FUNCTION_BLOCK MulticastTwoConCtl (* Composite Function Block Type *)
  (* Standard: 61499-2 *)
  (* Version 0.2, 2003-12-05, JHC, Rockwell Automation, Renamed from NEWCOMPFB. *)
  (* Version 0.1, 2002-01-08, JHC, Rockwell Automation, Added DLY FB as example. *)
  (* Version 0.0, 2000-05-27, JHC, Rockwell Automation *)
  (* Compiler header: package fb.rt.cs725; *)
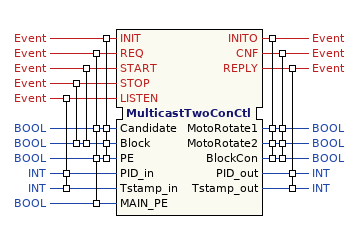
  EVENT_INPUT
    INIT WITH Candidate, Block, PE; (* Initialization Request *)
    REQ WITH Candidate, PE, MAIN_PE; (* Normal Execution Request *)
    START WITH Block;
    STOP WITH Block;
    LISTEN WITH Tstamp_in, PID_in;
  END_EVENT
  EVENT_OUTPUT
    INITO WITH MotoRotate1, MotoRotate2, BlockCon; (* Initialization Confirm *)
    CNF WITH MotoRotate1, MotoRotate2, BlockCon; (* Execution Confirmation *)
    REPLY WITH PID_out, Tstamp_out;
  END_EVENT
  VAR_INPUT
    Candidate : BOOL;
    Block : BOOL;
    PE : BOOL;
    PID_in : INT;
    Tstamp_in : INT;
    MAIN_PE : BOOL;
  END_VAR
  VAR_OUTPUT
    MotoRotate1 : BOOL;
    MotoRotate2 : BOOL;
    BlockCon : BOOL;
    PID_out : INT;
    Tstamp_out : INT;
  END_VAR
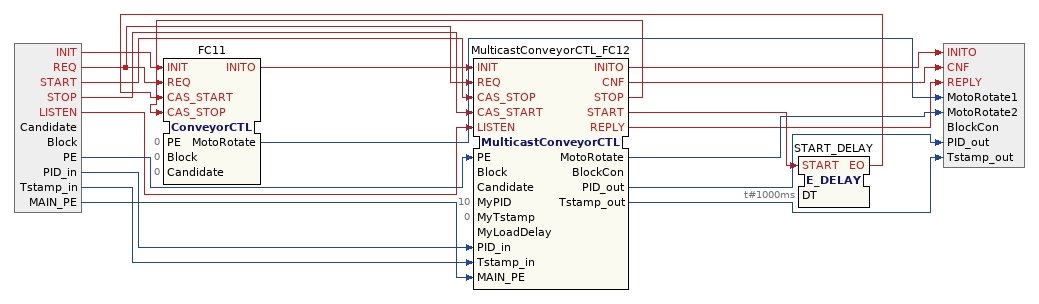
  FBS
    FC11 : ConveyorCTL(PE := 0, Block := 0, Candidate := 0);
    MulticastConveyorCTL_FC12 : MulticastConveyorCTL(MyPID := 10, MyTstamp := 0);
    START_DELAY : E_DELAY(DT := t#1000ms);
  END_FBS
  EVENT_CONNECTIONS
    INIT TO FC11.INIT;
    REQ TO FC11.REQ;
    LISTEN TO MulticastConveyorCTL_FC12.LISTEN;
    MulticastConveyorCTL_FC12.REPLY TO REPLY;
    FC11.INITO TO MulticastConveyorCTL_FC12.INIT;
    MulticastConveyorCTL_FC12.CNF TO CNF;
    MulticastConveyorCTL_FC12.INITO TO INITO;
    START TO MulticastConveyorCTL_FC12.CAS_STOP;
    STOP TO MulticastConveyorCTL_FC12.CAS_START;
    REQ TO MulticastConveyorCTL_FC12.REQ;
    MulticastConveyorCTL_FC12.START TO START_DELAY.START;
    START_DELAY.EO TO FC11.CAS_START;
    MulticastConveyorCTL_FC12.STOP TO FC11.CAS_STOP;
  END_CONNECTIONS
  DATA_CONNECTIONS
    FC11.MotoRotate TO MotoRotate1;
    PE TO MulticastConveyorCTL_FC12.PE;
    PID_in TO MulticastConveyorCTL_FC12.PID_in;
    Tstamp_in TO MulticastConveyorCTL_FC12.Tstamp_in;
    MulticastConveyorCTL_FC12.Tstamp_out TO Tstamp_out;
    MulticastConveyorCTL_FC12.PID_out TO PID_out;
    MulticastConveyorCTL_FC12.MotoRotate TO MotoRotate2;
    MAIN_PE TO MulticastConveyorCTL_FC12.MAIN_PE;
  END_CONNECTIONS
END_FUNCTION_BLOCK
